// TIA Portal V17 export
// export: Created 2025-03-05T08:03:41.479385Z, ExportSetting WithDefaults, DisplayName Totally Integrated Automation Portal, DisplayVersion V17 Update 8, DisplayName TIA Portal Openness, DisplayVersion V17 Update 8, DisplayName TIA Portal Version Control Interface, DisplayVersion V17, DisplayName SINAMICS Startdrive Advanced, DisplayVersion V17 SP2, DisplayName SINAMICS Startdrive G110M, G120, G120C, G120D, G120P, G115D, DisplayVersion V17 SP2, DisplayName SINAMICS Startdrive G130, G150, S120, S150, SINAMICS MV, S210, DisplayVersion V17 SP2, DisplayName STEP 7 Professional, DisplayVersion V17 Update 8, DisplayName SINUMERIK ONE STEP 7 Toolbox, DisplayVersion V17 Update 12, DisplayName SINUMERIK 840D sl STEP 7 Toolbox, DisplayVersion V17 Update 12, DisplayName STEP 7 Safety, DisplayVersion V17 Update 6, DisplayName WinCC Advanced, DisplayVersion V17 Update 8
TYPE "POWDER SWITCH"
// stored: IsFailsafeCompliant false
   STRUCT
      "Hopper 1 General Conditions" : Bool;   // Hopper 1 General Conditions
      "Hopper 1 Initial Conditions" : Bool;   // Hopper 1 Initial Conditions
      "Hopper 1 Manual Request" : Bool;   // Hopper 1 Manual Request
      "Hopper 1 Auto Request" : Bool;   // Hopper 1 Auto Request
      "Hopper 1 Global Request" : Bool;   // Hopper 1 Global Request
      "Hopper 1 Command" : Bool;   // Hopper 1 Command
      "Hopper 1" : Bool;   // Hopper 1
      "Feedback Hopper 1" : Bool;   // Feedback Hopper 1
      "Hopper 2 General Conditions" : Bool;   // Hopper 2 General Conditions
      "Hopper 2 Initial Conditions" : Bool;   // Hopper 2 Initial Conditions
      "Hopper 2 Manual Request" : Bool;   // Hopper 2 Manual Request
      "Hopper 2 Auto Request" : Bool;   // Hopper 2 Auto Request
      "Hopper 2 Global Request" : Bool;   // Hopper 2 Global Request
      "Hopper 2 Command" : Bool;   // Hopper 2 Command
      "Hopper 2" : Bool;   // Hopper 2
      "Feedback Hopper 2" : Bool;   // Feedback Hopper 2
      "Hopper 1 General Conditions Help" : Bool;   // Hopper 1 General Conditions Help
      "Hopper 1 Initial Conditions Help" : Bool;   // Hopper 1 Initial Conditions Help
      "Hopper 2 General Conditions Help" : Bool;   // Hopper 2 General Conditions Help
      "Hopper 2 Initial Conditions Help" : Bool;   // Hopper 2 Initial Conditions Help
   END_STRUCT;
END_TYPE
